FUNCTION_BLOCK FB_Machine EXTENDS FB_PackML_BaseModule
VAR
	Boiler		: 	I_Boiler;
	Dispenser	: 	I_Dispenser;
END_VAR

{warning 'Add method implementation '}
METHOD CyclicLogic
END_METHOD

END_FUNCTION_BLOCK

(* stored: Version 1.1.0.1
   POU FB_Machine: Id {66cd1380-c52f-4694-bc09-18455997d862}, SpecialFunc None
   Method CyclicLogic: Id {041eac44-05ea-481d-bf59-fdcc1dd5374b} *)
